# EPICS autosave request: utcaApp/Db/trigger_mux_channel.req
$(P)$(R)$(TRIGGER_NAME)$(TRIGGER_CHAN)$(TRIGGER_DIR)Src-Sel
$(P)$(R)$(TRIGGER_NAME)$(TRIGGER_CHAN)$(TRIGGER_DIR_SEL)Sel-SP
